Universal Robots URScript: 5.12.2024.script

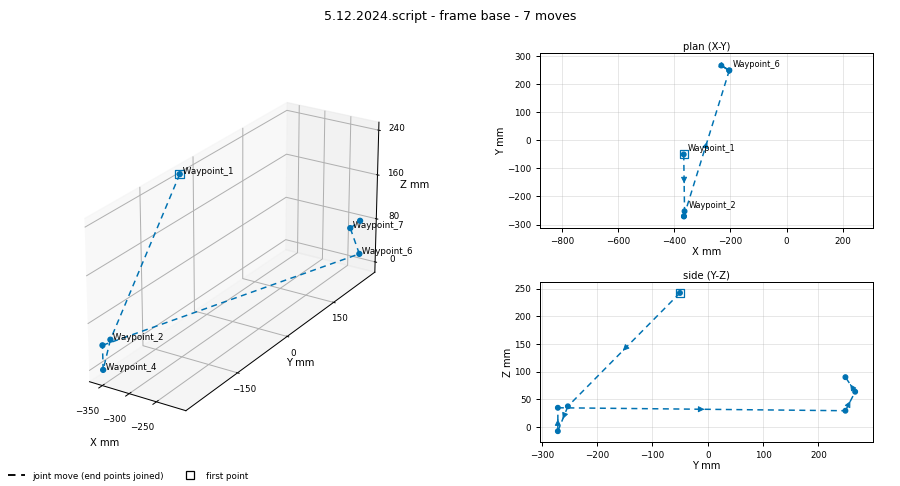
[picture p0: tool path of 5.12.2024.script in frame base, 7 of 7 moves have a stored position in this frame; points joined in program order, loops and branches not executed]
def P5122024():
  set_safety_mode_transition_hardness(1)
  set_tool_voltage(24)
  set_gravity([0.0, 0.0, 9.82])
  set_tcp(p[0.0375,0.0,0.083,0.0,0.0,0.0])
  set_payload(1.0, [-0.012, -0.005, 0.046])
  set_standard_analog_input_domain(0, 1)
  set_standard_analog_input_domain(1, 1)
  set_tool_analog_input_domain(0, 1)
  set_tool_analog_input_domain(1, 1)
  set_analog_outputdomain(0, 0)
  set_analog_outputdomain(1, 0)
  set_input_actions_to_default()
  step_count_893c2823_e373_482f_b399_449265bbbe33 = 0.0
  thread Step_Counter_Thread_edfdbf7e_928d_4bb1_98bc_e84468c5d915():
    while (True):
      step_count_893c2823_e373_482f_b399_449265bbbe33 = step_count_893c2823_e373_482f_b399_449265bbbe33 + 1.0
      sync()
    end
  end
  run Step_Counter_Thread_edfdbf7e_928d_4bb1_98bc_e84468c5d915()
  global parallelo=p[1.2122131398326075E-6,0.1500036957322406,0.2000145501490997,8.665644107087391E-5,-3.074787590163792E-5,2.4958435593227474E-5]
  global perpendicolare=p[1.3133400607635848E-5,0.4499782418304641,0.014952299880116995,4.8195394996186283E-4,2.221762010521941,2.2210105916999128]
  rtde_set_watchdog("speed_slider_mask", 10.0, "ignore")
  # begin: URCap Installation Node
  #   Source: OnRobot, 6.1.0, OnRobot A/S
  #   Type: OnRobot Setup
  # end: URCap Installation Node
  $ 1 "BeforeStart"
  $ 2 "MoveJ"
  $ 3 "Waypoint_1" "breakAfter"
  movej(get_inverse_kin(p[-.366564742567, -.050190250743, .242410149702, -.456025890705, -2.994706259561, .070170829900], qnear=[-2.606410090123312, -1.5642054716693323, -1.591473404561178, -1.438688103352682, 1.5364649295806885, -38.42861863768386]), a=1.3962634015954636, v=1.0471975511965976)
  while (True):
    $ 4 "Robot Program"
    $ 5 "MoveJ"
    $ 6 "Waypoint_2" "breakAfter"
    movej(get_inverse_kin(p[-.363667383712, -.252721442625, .037530635500, .144353083856, -3.114008582285, .019594089015], qnear=[-2.2134159247027796, -2.2273600737201136, -1.661717716847555, -0.7957523504840296, 1.5568493604660034, -38.42870208418655]), a=1.3962634015954636, v=1.0471975511965976)
    $ 7 "Waypoint_4" "breakAfter"
    movej(get_inverse_kin(p[-.365903057087, -.270898156432, -.007466767740, -.424167002271, 3.111861554192, -.010715512125], qnear=[-2.2096059958087366, -2.3929670492755335, -1.596741024647848, -0.7158835569964808, 1.5721138715744019, -38.603549687030785]), a=1.3962634015954636, v=1.0471975511965976)
    $ 8 "Waypoint_5" "breakAfter"
    movej(get_inverse_kin(p[-.365911420572, -.270852364203, .034885578493, -.423983942939, 3.111861250996, -.010563360473], qnear=[-2.209653679524557, -2.271116558705465, -1.575083080922262, -0.859476391469137, 1.572797417640686, -38.60316535628127]), a=1.3962634015954636, v=1.0471975511965976)
    $ 9 "Waypoint_6" "breakAfter"
    movej(get_inverse_kin(p[-.204329076825, .248851181414, .029521370449, -1.648072110986, -2.642272822520, .003031129057], qnear=[-3.5972164312945765, -1.8973410765277308, -2.355333391820089, -0.4296467939959925, 1.5685527324676514, -38.602456776264184]), a=1.3962634015954636, v=1.0471975511965976)
    $ 10 "Waypoint_7" "breakAfter"
    movej(get_inverse_kin(p[-.232573555161, .266464524885, .063846143105, -1.404591129372, -2.151653187794, -.837292867860], qnear=[-3.2194324175464075, -2.0968430677997034, -2.5493343512164515, 0.04776346683502197, 0.8103605508804321, -38.22981664336013]), a=1.3962634015954636, v=1.0471975511965976)
    $ 11 "Waypoint_8" "breakAfter"
    movej(get_inverse_kin(p[-.204365607437, .248866595892, .090178337514, -1.648118148134, -2.642142373003, .003135321499], qnear=[-3.597408119832174, -1.6314314047442835, -2.2459853331195276, -0.8048031965838831, 1.5708428621292114, -38.602936951282494]), a=1.3962634015954636, v=1.0471975511965976)
  end
end
